FUNCTION_BLOCK ATV320_HMI (* Service Interface Function Block Type *)
  (* Standard: 61499-2 *)
  (* Version 0.0, 06/08/2021, SESA371406, Schneider Electric, template *)
  PACKAGE SE.Nereda;
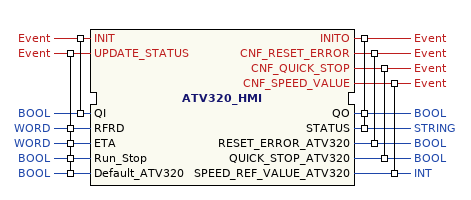
  EVENT_INPUT
    INIT WITH QI;
    UPDATE_STATUS WITH RFRD, ETA, Run_Stop, Default_ATV320;
  END_EVENT
  EVENT_OUTPUT
    INITO WITH QO, STATUS;
    CNF_RESET_ERROR WITH RESET_ERROR_ATV320;
    CNF_QUICK_STOP WITH QUICK_STOP_ATV320;
    CNF_SPEED_VALUE WITH SPEED_REF_VALUE_ATV320;
  END_EVENT
  VAR_INPUT
    QI : BOOL;
    RFRD : WORD; (* ACTUAL_SPEED_VALUE *)
    ETA : WORD; (* STATUE_WORD *)
    Run_Stop : BOOL;
    Default_ATV320 : BOOL;
  END_VAR
  VAR_OUTPUT
    QO : BOOL; (* Event Output Qualifier *)
    STATUS : STRING; (* Service Status *)
    RESET_ERROR_ATV320 : BOOL;
    QUICK_STOP_ATV320 : BOOL;
    SPEED_REF_VALUE_ATV320 : INT;
  END_VAR
  SERVICE /
    SEQUENCE 
    END_SEQUENCE
  END_SERVICE
END_FUNCTION_BLOCK
